FUNCTION_BLOCK FB_HMI
VAR_INPUT
END_VAR
VAR_OUTPUT
END_VAR
VAR

stHMI_In    : stHMI_In;
stHMI_Out   : stHMI_Out;






    

END_VAR

M_Inputs();
M_Outputs();

METHOD M_Inputs : BOOL
VAR_INPUT
END_VAR
// User Speed/Override Settings

fbCNC.fChannelOverride := stHMI_In.fChannelOverride;
END_METHOD

METHOD M_Outputs : BOOL
VAR_INPUT
END_VAR
// Limit and Homing Switch Mapping

stHMI_Out.bX1HomeSwitch := fbCNC.bXHomingSwitch;	
stHMI_Out.bX2HomeSwitch := fbCNC.bX2HomingSwitch;
stHMI_Out.bXLimitSwitch := fbCNC.bXLimitSwitch;	
stHMI_Out.bYHomeSwitch := fbCNC.bYHomingSwitch;
stHMI_Out.bYLimitSwitch := fbCNC.bYLimitSwitch;	
stHMI_Out.bZHomeSwitch  := fbCNC.bZHomingSwitch;	

// Interpreter Channel State

stHMI_Out.sInterpreterState := TO_STRING(fbNCInfo.eInterpreterState);

// Channel Override Speed

stHMI_Out.fChannelOverrideSpeed := fbCNC.fChannelOverride;

// Axis Status

stHMI_Out.bXAxisHomed:= fbCNC.X_Ref.Status.Homed;
stHMI_Out.bX2AxisHomed:= fbCNC.X2_Ref.Status.Homed;
stHMI_Out.bYAxisHomed:= fbCNC.Y_Ref.Status.Homed;
stHMI_Out.bZAxisHomed:= fbCNC.Z_Ref.Status.Homed;

// Position

stHMI_Out.fActPosX := fbCNC.X_Ref.NcToPlc.ActPos;
stHMI_Out.fActPosX2 := fbCNC.X2_Ref.NcToPlc.ActPos;
stHMI_Out.fActPosY := fbCNC.Y_Ref.NcToPlc.ActPos;
stHMI_Out.fActPosZ := fbCNC.Z_Ref.NcToPlc.ActPos;
END_METHOD

END_FUNCTION_BLOCK

(* stored: Version 1.1.0.1, ProductVersion 3.1.4024.9
   POU FB_HMI: Id {74169dc0-8ac6-4a2f-90d1-a2b9ba1bf1ca}, SpecialFunc None
   Method M_Inputs: Id {14d1c6a3-722d-4790-a5a9-7e9d7bd7fdb8}
   Method M_Outputs: Id {3525acce-6037-42c8-9504-c0bff51f5c6e} *)
